PROGRAM MAIN
VAR
END_VAR

END_PROGRAM

(* stored: Version 1.1.0.1
   POU MAIN: Id {1195c322-cb2a-4373-bccb-ec4abdef93b4} *)
